FUNCTION_BLOCK FB_NestedView
VAR_INPUT CONSTANT
	View		: FB_BA_View;
		Enable	: FB_BA_BV_Op := (
					iParent			:= View,
					iProfile		:= MyProfiles.BVOp_Prf,
					bValueRm		:= FALSE
				);		
		Value	: FB_BA_AV_Op := (
					iParent			:= View,
					iProfile		:= MyProfiles.AVOp_Prf,
					fValueRm		:= 0.0
				);	
END_VAR

View();
Enable();
Value();

END_FUNCTION_BLOCK

(* stored: Version 1.1.0.1, ProductVersion 3.1.4024.5
   POU FB_NestedView: Id {0c57493a-b28c-4808-ac95-a2a244c7d8a3}, SpecialFunc None *)
